// TwinCAT 3 PLC project Sample
// ProgramVersion: 3.1.4024.0
// libraries:
//   Tc2_Standard, * (Beckhoff Automation GmbH)
//   Tc2_System, * (Beckhoff Automation GmbH)
//   Tc3_Module, * (Beckhoff Automation GmbH)
// project tree:
//   / PlcTask.TcTTO
//   POUs/ MAIN.TcPOU
// real-time tasks:
//   TASK PlcTask: cycle T#10ms, priority 20, ADS port 350

CONFIGURATION Sample
    RESOURCE PLC ON TwinCAT3
        TASK PlcTask(INTERVAL := T#10ms, PRIORITY := 20);
        PROGRAM MAIN WITH PlcTask : MAIN;
    END_RESOURCE
END_CONFIGURATION

// ---- POUs/MAIN.TcPOU
PROGRAM MAIN
VAR
	n_cnt_1 : UINT;
	n_cnt_2 : UINT;
	n_cnt_3 : UINT;
	
	ton_1 : TON := (PT := T#0.2S);
	ton_2 : TON := (PT := T#0.5S);
	ton_3 : TON := (PT := T#1S);
END_VAR

ton_1(IN := NOT ton_1.Q);
ton_2(IN := NOT ton_2.Q);
ton_3(IN := NOT ton_3.Q);

IF ton_1.Q THEN
	n_cnt_1 := n_cnt_1 + 1;
END_IF

IF ton_2.Q THEN
	n_cnt_2 := n_cnt_2 + 1;
END_IF

IF ton_3.Q THEN
	n_cnt_3 := n_cnt_3 + 1;
END_IF

END_PROGRAM
